# EPICS substitutions: evgMrmApp/Db/NSLS/vme-evg230-nsls2.substitutions
file evgAcTrig.db {
pattern { P, OBJ }
{ "$(SYS){$(D)-AcTrig}", "$(EVG):AcTrig" }
}

file evgDbus.db {
pattern { P, OBJ, EVG, dbusBit }
{ "$(SYS){$(D)-Dbus:0}", "$(EVG):Dbus0", $(EVG), 0 }
{ "$(SYS){$(D)-Dbus:1}", "$(EVG):Dbus1", $(EVG), 1 }
{ "$(SYS){$(D)-Dbus:2}", "$(EVG):Dbus2", $(EVG), 2 }
{ "$(SYS){$(D)-Dbus:3}", "$(EVG):Dbus3", $(EVG), 3 }
{ "$(SYS){$(D)-Dbus:4}", "$(EVG):Dbus4", $(EVG), 4 }
{ "$(SYS){$(D)-Dbus:5}", "$(EVG):Dbus5", $(EVG), 5 }
{ "$(SYS){$(D)-Dbus:6}", "$(EVG):Dbus6", $(EVG), 6 }
{ "$(SYS){$(D)-Dbus:7}", "$(EVG):Dbus7", $(EVG), 7 }
}

file evgEvtClk.db {
pattern { P, OBJ}
{"$(SYS){$(D)-EvtClk}", "$(EVG):EvtClk"}
}

file evgInput.db {
pattern { P, OBJ, , SYS, D, Num }
{ "$(SYS){$(D)-Inp:Front0}", "$(EVG):FrontInp0", $(SYS), $(D), 0 }
{ "$(SYS){$(D)-Inp:Front1}", "$(EVG):FrontInp1", $(SYS), $(D), 1 }
{ "$(SYS){$(D)-Inp:Univ0}",  "$(EVG):UnivInp0",  $(SYS), $(D), 2 }
{ "$(SYS){$(D)-Inp:Univ1}",  "$(EVG):UnivInp1",  $(SYS), $(D), 3 }
{ "$(SYS){$(D)-Inp:Univ2}",  "$(EVG):UnivInp2",  $(SYS), $(D), 4 }
{ "$(SYS){$(D)-Inp:Univ3}",  "$(EVG):UnivInp3",  $(SYS), $(D), 5 }
}

file evgMrm.db {
pattern { P, OBJ,  EVG }
{ "$(SYS){$(D)}", $(EVG), $(EVG) }
}

file evgMxc.db {
pattern { P, OBJ, SYS, D }
{ "$(SYS){$(D)-Mxc:0}", "$(EVG):Mxc0", $(SYS), $(D) }
{ "$(SYS){$(D)-Mxc:1}", "$(EVG):Mxc1", $(SYS), $(D) }
{ "$(SYS){$(D)-Mxc:2}", "$(EVG):Mxc2", $(SYS), $(D) }
{ "$(SYS){$(D)-Mxc:3}", "$(EVG):Mxc3", $(SYS), $(D) }
{ "$(SYS){$(D)-Mxc:4}", "$(EVG):Mxc4", $(SYS), $(D) }
{ "$(SYS){$(D)-Mxc:5}", "$(EVG):Mxc5", $(SYS), $(D) }
{ "$(SYS){$(D)-Mxc:6}", "$(EVG):Mxc6", $(SYS), $(D) }
{ "$(SYS){$(D)-Mxc:7}", "$(EVG):Mxc7", $(SYS), $(D) }
}

file evgOutput.db {
pattern { P, OBJ }
{ "$(SYS){$(D)-Out:Front0}", "$(EVG):FrontOut0" }
{ "$(SYS){$(D)-Out:Front1}", "$(EVG):FrontOut1" }
{ "$(SYS){$(D)-Out:Front2}", "$(EVG):FrontOut2" }
{ "$(SYS){$(D)-Out:Front3}", "$(EVG):FrontOut3" }
}

file evgSoftEvt.db {
pattern { P, OBJ }
{ "$(SYS){$(D)-SoftEvt}", "$(EVG):SoftEvt" }
}

file evgSoftSeq.db {
pattern { P, EVG, seqNum, NELM, ASGUSER }
{ "$(SYS){$(D)-SoftSeq:0}",  $(EVG), 0, 2047, "OPERATOR" }
{ "$(SYS){$(D)-SoftSeq:1}", $(EVG), 1, 2047, "OPERATOR" }
{ "$(SYS){$(D)-SoftSeq:2}",  $(EVG), 2, 2047, "OPERATOR" }
{ "$(SYS){$(D)-SoftSeq:3}", $(EVG), 3, 2047, "OPERATOR" }
pattern { P, EVG, seqNum, NELM, ENALNK }
{ "$(SYS){$(D)-SoftSeq:Inj}",  $(EVG), 4, 2047, "$(SYS){$(D)-SSC}Inject:B-Calc_" }
{ "$(SYS){$(D)-SoftSeq:InjN}",  $(EVG), 5, 2047, "$(SYS){$(D)-SSC}Inject:N-Calc_" }
}

file nsls2-inj-ssc.db {
{P="$(SYS){$(D)-SSC}",
 SYS="\$(SYS)", D="\$(D)",
 SEQN="InjN", SEQB="Inj",
}
}

file evgTrigEvt.db {
pattern { P, OBJ, EVG, trigEvtNum }
{ "$(SYS){$(D)-TrigEvt:0}", "$(EVG):TrigEvt0", $(EVG), 0 }
{ "$(SYS){$(D)-TrigEvt:1}", "$(EVG):TrigEvt1", $(EVG), 1 }
{ "$(SYS){$(D)-TrigEvt:2}", "$(EVG):TrigEvt2", $(EVG), 2 }
{ "$(SYS){$(D)-TrigEvt:3}", "$(EVG):TrigEvt3", $(EVG), 3 }
{ "$(SYS){$(D)-TrigEvt:4}", "$(EVG):TrigEvt4", $(EVG), 4 }
{ "$(SYS){$(D)-TrigEvt:5}", "$(EVG):TrigEvt5", $(EVG), 5 }
{ "$(SYS){$(D)-TrigEvt:6}", "$(EVG):TrigEvt6", $(EVG), 6 }
{ "$(SYS){$(D)-TrigEvt:7}", "$(EVG):TrigEvt7", $(EVG), 7 }
}

file databuftx.db
{pattern
{ P, OBJ, PROTO }
{ "$(SYS){$(D)}", "$(EVG):BUFTX", 1 }
}

file "databuftxCtrl.db"
{pattern
{ P, OBJ }
{ "$(SYS){$(D)}", "$(EVG):BUFTX" }
}
